(* IEC 61131-3 sources: JaccoSigma/tempclass/Class/Virtual_User, 1 file *)

(* ---- Virtual_User.st ---- *)
(*!
<Class
	Name               = "Virtual_User"
	Revision           = "1.0"
	RealtimeTask       = "false"
	CyclicTask         = "false"
	BackgroundTask     = "false"
	Sigmatek           = "true"
	OSInterface        = "false"
	HighPriority       = "false"
	Automatic          = "false"
	UpdateMode         = "Prescan"
	IconPath           = ".\Class\Virtual_User\toolbox.ICO"
	SharedCommandTable = "true"
	Objectsize         = "(284,120)"
	Comment            = "V1.0 Interface of user&#13;&#10;have some global user methods&#13;&#10;(AppliStart, AppliRun, ...)&#13;&#10;these functions are called by _ET_Runtime.">
	<Channels>
		<Server Name="Server0" Visualized="true" Initialize="false" WriteProtected="false" Retentive="false" Comment="if you want to use this class connect this server to the client &quot;Application&quot; of _Et_Runtime"/>
	</Channels>
</Class>
*)
Virtual_User : CLASS
  //Servers:
	Server0 	: SvrChCmd_DINT;
  //Clients:
  //Variables:
  //Functions:
				//! <Function Comment="function is called during the start of the application&#13;&#10;" Name="AppliStart"/>
	FUNCTION VIRTUAL GLOBAL AppliStart;
				//! <Function Comment="function is called if the appli started successfull" Name="AppliReady"/>
	FUNCTION VIRTUAL GLOBAL AppliReady;
				//! <Function Comment="function is called, while the application runs" Name="AppliRun"/>
	FUNCTION VIRTUAL GLOBAL AppliRun;
				//! <Function Comment="the method doesn´t exist any more" Name="AppliEnd"/>
	FUNCTION VIRTUAL GLOBAL AppliEnd;
  //Tables:
	FUNCTION @STD
		VAR_OUTPUT
			ret_code	: CONFSTATES;
		END_VAR;
	FUNCTION GLOBAL TAB @CT_;
END_CLASS;

//*********************Inserted from .\Virtual_User\Virtual_User_00_00.st*********************

FUNCTION VIRTUAL GLOBAL Virtual_User::AppliStart

END_FUNCTION //VIRTUAL GLOBAL Virtual_User::AppliStart

FUNCTION VIRTUAL GLOBAL Virtual_User::AppliReady

END_FUNCTION //VIRTUAL GLOBAL Virtual_User::AppliReady

FUNCTION VIRTUAL GLOBAL Virtual_User::AppliRun

END_FUNCTION //VIRTUAL GLOBAL Virtual_User::AppliRun

FUNCTION VIRTUAL GLOBAL Virtual_User::AppliEnd

END_FUNCTION //VIRTUAL GLOBAL Virtual_User::AppliEnd
